// TIA Portal V18 export
DATA_BLOCK "L1_flyingCutoff"   // DB22
{ S7_Optimized_Access := 'TRUE' }
VERSION : 0.1
// stored: AutoNumber true, DBAccessibleFromOPCUA true, DBAccessibleFromWebserver true, IsOnlyStoredInLoadMemory false, IsRetainMemResEnabled false, IsWriteProtectedInAS false, MemoryReserve 100
   VAR RETAIN
      data : "LGasp_flyingCutoff";
   END_VAR
BEGIN
END_DATA_BLOCK
